# B&R Automation Studio project TrakBasisProject (part 2)

#### Set_Testcases.c
```c
/********************************************************************
 * COPYRIGHT --
 ********************************************************************
 * Program: -
 * Author:
 * Created:
 ********************************************************************
 * Tests for ...
 ********************************************************************/

#include <bur/plctypes.h>

#ifdef _DEFAULT_INCLUDES
#include <AsDefault.h>
#endif

#include "UnitTest.h"

_TEST waitForReadyForPowerOn (void)
{
	TEST_BUSY_CONDITION(0 == gTrakCtrl.Status.ReadyForPowerOn);
	TEST_ASSERT(gTrakCtrl.Status.ReadyForPowerOn);

	TEST_DONE;
}

_TEST waitForCommunicationReady (void)
{
	TEST_BUSY_CONDITION(0 == gTrakCtrl.Status.CommunicationReady);
	TEST_ASSERT(gTrakCtrl.Status.CommunicationReady);

	TEST_DONE;
}

_TEST waitForPLCopenStateDisabled (void)
{
	TEST_ASSERT(gTrakCtrl.Status.PLCopenState.Disabled);

	TEST_DONE;
}

_TEST setPowerOnAndCheckStatus (void)
{
	gTrakCtrl.Command.Power = 1;

	TEST_BUSY_CONDITION(0 == gTrakCtrl.Status.PowerOn);
	TEST_ASSERT(gTrakCtrl.Status.PowerOn);

	TEST_DONE;
}

_TEST waitForPLCopenStateReady (void)
{
	TEST_BUSY_CONDITION(0 == gTrakCtrl.Status.PLCopenState.Ready);
	TEST_ASSERT(gTrakCtrl.Status.PLCopenState.Ready);

	TEST_DONE;
}

_TEST setCommandMoveAbsolute (void)
{
	gTrakCtrl.Command.Move.Absolute = 1;
	gTrakCtrl.Parameter.Position = 0.0;
	gTrakCtrl.Parameter.Speed = 2.0;
	gTrakCtrl.Parameter.Acceleration = 20.0;
	gTrakCtrl.Parameter.Deceleration = 20.0;

	TEST_DONE;
}

_TEST waitForMovementAfterCommandMoveAbsolute (void)
{
	TEST_BUSY_CONDITION(1 == gTrakCtrl.Command.Move.Absolute);
	TEST_BUSY_CONDITION(0 == gTrakCtrl.Status.MovementDetected);
	TEST_ASSERT(gTrakCtrl.Status.MovementDetected);

	TEST_DONE;
}

_TEST waitForMovementAbsoluteStops (void)
{
	TEST_BUSY_CONDITION(1 == gTrakCtrl.Status.MovementDetected);
	TEST_ASSERT(0 == gTrakCtrl.Status.MovementDetected);
	TEST_DONE;
}

_TEST setCommandMoveVelocity (void)
{
	gTrakCtrl.Command.Move.Velocity = 1;
	gTrakCtrl.Parameter.Position = 0.0;
	gTrakCtrl.Parameter.Speed = 2.0;
	gTrakCtrl.Parameter.Acceleration = 20.0;
	gTrakCtrl.Parameter.Deceleration = 20.0;

	TEST_DONE;
}

_TEST waitForMovementAfterCommandMoveVelocity (void)
{
	TEST_BUSY_CONDITION(1 == gTrakCtrl.Command.Move.Velocity);
	TEST_BUSY_CONDITION(0 == gTrakCtrl.Status.MovementDetected);

	TEST_ASSERT(gTrakCtrl.Status.MovementDetected);

	TEST_DONE;
}

_TEST checkActualSpeedAfterCommandMoveVelocity (void)
{
	TEST_BUSY_CONDITION(2.0 > gTrakCtrl.Status.Shuttle[1].ActVelocity);

	TEST_ASSERT(gTrakCtrl.Status.Shuttle[1].Valid);
	TEST_ASSERT_REAL_WITHIN(0.1, 2.0, gTrakCtrl.Status.Shuttle[1].ActVelocity);
	TEST_ASSERT_EQUAL_STRING("Sector_1", gTrakCtrl.Status.Shuttle[1].ActSector);

	TEST_DONE;
}

_TEST setCommandHalt (void)
{
	gTrakCtrl.Command.Move.Halt = 1;

	TEST_DONE;
}

_TEST waitForMovementStopsAfterCommandHalt (void)
{
	TEST_BUSY_CONDITION(1 == gTrakCtrl.Command.Move.Halt);
	TEST_BUSY_CONDITION(1 == gTrakCtrl.Status.MovementDetected);

	TEST_ASSERT(0 == gTrakCtrl.Status.MovementDetected);
	TEST_ASSERT(gTrakCtrl.Status.Shuttle[1].Valid);
	TEST_ASSERT_EQUAL_REAL(0.0, gTrakCtrl.Status.Shuttle[1].ActVelocity);
	TEST_ASSERT_EQUAL_STRING("Sector_1", gTrakCtrl.Status.Shuttle[1].ActSector);

	TEST_DONE;
}

/*
B+R UnitTest: This is generated code.
Do not edit! Do not move!
Description: UnitTest Testprogramm infrastructure (TestSet).
LastUpdated: 2025-09-17 11:53:31Z
By B+R UnitTest Helper Version: 2.0.0.0
*/
UNITTEST_FIXTURES(fixtures)
{
	new_TestFixture("waitForReadyForPowerOn", waitForReadyForPowerOn),
	new_TestFixture("waitForCommunicationReady", waitForCommunicationReady),
	new_TestFixture("waitForPLCopenStateDisabled", waitForPLCopenStateDisabled),
	new_TestFixture("setPowerOnAndCheckStatus", setPowerOnAndCheckStatus),
	new_TestFixture("waitForPLCopenStateReady", waitForPLCopenStateReady),
	new_TestFixture("setCommandMoveAbsolute", setCommandMoveAbsolute),
	new_TestFixture("waitForMovementAfterCommandMoveAbsolute", waitForMovementAfterCommandMoveAbsolute),
	new_TestFixture("waitForMovementAbsoluteStops", waitForMovementAbsoluteStops),
	new_TestFixture("setCommandMoveVelocity", setCommandMoveVelocity),
	new_TestFixture("waitForMovementAfterCommandMoveVelocity", waitForMovementAfterCommandMoveVelocity),
	new_TestFixture("checkActualSpeedAfterCommandMoveVelocity", checkActualSpeedAfterCommandMoveVelocity),
	new_TestFixture("setCommandHalt", setCommandHalt),
	new_TestFixture("waitForMovementStopsAfterCommandHalt", waitForMovementStopsAfterCommandHalt),
};

UNITTEST_CALLER_COMPLETE_EXPLICIT(Set_Testcases, "Set_Testcases", 0, 0, fixtures, 0, 0, 0);
```

### Library Logical/UnitTest/Libraries/UnitTest (ANSIC, version 6.3.0) - Static library for UnitTest programs written in ANSI C /C++

#### UnitTest.h
```c
/*****************************************************************************
 * COPYRIGHT (C) BERNECKER + RAINER
 *****************************************************************************
 * Library:  UnitTest
 * File:     UnitTest.h
 * Author:   B+R
 *****************************************************************************
 * Description: Static library for UnitTest programs written in ANSI C /C++
 *
 * Add the path "\Logical\TS_UnitTest\Libraries\UnitTest\" to the
 * "Additional include directories" in the tab "Build" (PLC Properties)
 ******************************************************************************/

#ifndef	__UNITTEST_H__
#define	__UNITTEST_H__
#ifdef __cplusplus
extern "C"
{
#endif
#include <bur/plctypes.h>

#ifndef NULL
#define	NULL	0
#endif
#include "include/Test.h"

#include "include/TestCase.h"
#include "include/TestListener.h"
#include "include/TestResult.h"
#include "include/TestCaller.h"

#include "include/AssertImpl.h"
#include "include/HelperMacro.h"
#include "include/utRunner.h"

/* function is a test case */
#define _TEST 			static testStatusEnum

/* function is a setup */
#define _SETUP_TEST 	static testStatusEnum 	setupTest

/* function is a teardown */
#define _TEARDOWN_TEST 	static testStatusEnum 	teardownTest

/* function is a setup for whole test set */
#define _SETUP_SET		static testStatusEnum	setupSet

/* function is a teardown for whole test set */
#define _TEARDOWN_SET 	static testStatusEnum	teardownSet

/* function is a cyclic handler for test set */
#define _CYCLIC_SET		static void 			cyclicSetCaller

/* Skipped test case */
#define SKIP_TEST  		_TEST
/* Skip all test cases of set */
#define SKIP_TEST_SET

/* Dummies for smart edit autocompletion.
See AssertImpl.h for real macros used by the compiler  */
#ifdef _SMART_EDIT_DUMMY_

/* String comparison.
Returns true if the strings are equal. */
BOOL TEST_ASSERT_EQUAL_STRING(char *expected,char  *actual);
/* Wstring comparison.
Returns true if the WSTRINGS are equal. */
BOOL TEST_ASSERT_EQUAL_WSTRING(unsigned short *expected,unsigned short *actual);
 /* Compares two memory blocks.
Returns true if [size] bytes are equal. */
BOOL TEST_ASSERT_EQUAL_MEM(void *expected, void *actual,UDINT size);
/* Compares integer values. Usable for all integer types.
Avoid comparison of unsigned with signed types.
Returns true if they are equal.
Note: If different, values are reported as DINT values in the test report */
BOOL TEST_ASSERT_EQUAL_INT(expected, actual);

/* Compares REAL values with delta = (expected * TEST_FLOAT_PRECISION).
Returns true if (difference <= delta) */
BOOL TEST_ASSERT_EQUAL_REAL(REAL expected,REAL actual);
/* Compares REAL values with explicit delta.
Returns true if (difference <= delta) */
BOOL TEST_ASSERT_REAL_WITHIN(REAL delta, REAL expected, REAL actual);
/* Compares LREAL values with delta = (expected * TEST_DOUBLE_PRECISION).
Returns true if (difference <= delta) */
BOOL TEST_ASSERT_EQUAL_LREAL(LREAL expected,LREAL  actual);
/* Compares LREAL values with explicit delta.
Returns true if (difference <= delta) */
BOOL TEST_ASSERT_LREAL_WITHIN(LREAL delta, LREAL expected, LREAL actual);

/* Compares float values with delta = (expected * TEST_FLOAT_PRECISION).
Returns true if (difference <= delta) */
BOOL TEST_ASSERT_EQUAL_FLOAT(float expected, float actual);
/* Compares float values with explicit delta.
Returns true if (difference <= delta) */
BOOL TEST_ASSERT_FLOAT_WITHIN(float delta, float expected, float actual);
/* Compares double values with delta = (expected * TEST_DOUBLE_PRECISION).
Returns true if (difference <= delta) */
BOOL TEST_ASSERT_EQUAL_DOUBLE(double expected, double actual);
/* Compares double values with explicit delta.
Returns true if (difference <= delta) */
BOOL TEST_ASSERT_DOUBLE_WITHIN(double delta, double expected, double actual);

/* Returns true if pointer is null */
BOOL TEST_ASSERT_NULL(void *pointer);
/* Returns true if pointer is not null */
BOOL TEST_ASSERT_NOT_NULL(void *pointer);
/* Returns true, if condition evals to  true */
BOOL TEST_ASSERT_MESSAGE(condition, char *message);
/* Returns true, if condition evals to  true */
BOOL TEST_ASSERT(condition);

/* Returns always false */
BOOL TEST_FAIL(char *message);

/* Add a note to the test report */
void TEST_INFO(char *message);
/* Add a note with location information to the test report */
void TEST_INFO_POS(char *message);

#ifdef __cplusplus
/* Test if expression throws given exception.
Catches all other exceptions as failure.
Note: Available for C++ only */
void TEST_ASSERT_THROW(expression, type);

/* Fails if expression throws any exceptions.
Note: Available for C++ only*/
void TEST_ASSERT_NO_THROW(expression);
#endif

/* Adds a test function with description to the Testfixture.
See UNITTEST_FIXTURES() */
void new_TestFixture(char *name, _TEST function);

/* Adds a test function with description to the Testfixture.
This test will be skipped
See UNITTEST_FIXTURES() */
void skipTestFixture(char *name, _TEST function);

/* Defines the order of test cases.
Should look like this
UNITTEST_FIXTURES(fixtures)
{
	new_TestFixture("test_1",test_1),
	new_TestFixture("test_2",test_2),
	new_TestFixture("test_3",test_3)
}
*/
void UNITTEST_FIXTURES(fixtures)

/* Standard UnitTest caller without any setup / teardown methods*/
void UNITTEST_CALLER_TEST(caller, char *name, fixtures);

/* Standard UnitTest caller with macro setup / teardown for tests*/
void UNITTEST_CALLER_BASIC(caller, char *name, fixtures);

/* UnitTest caller with macro setup / teardown for tests and test set */
void UNITTEST_CALLER_SET(caller, char *name, fixtures);

/* UnitTest caller with macro setup / teardown for tests and test set and cylic*/
void UNITTEST_CALLER_COMPLETE(caller, char *name, fixtures);

/* UnitTest caller with explicit setup / teardown for suite */
void UNITTEST_CALLER_SET_EXPLICIT(caller,name,setupTest,teardownTest,fixtures, setupSuite, teardownSuite);

/* UnitTest caller with explicit setup / teardown for suite and cylic */
void UNITTEST_CALLER_COMPLETE_EXPLICIT(caller,name,setupTest,teardownTest,fixtures, setupSuite, teardownSuite, cyclicCaller);

/* Adds a test set with description to the fixture of test sets.
See UNITTEST_TESTSET_FIXTURES() */
void new_TestSet(testcaller);

/* Defines the order of test sets.
Should look like this
UNITTEST_TESTSET_FIXTURES(fixtures)
{
	new_TestSet(testSet_1),
	new_TestSet(testSet_2),
	new_TestSet(testSet_3)
}*/
void UNITTEST_TESTSET_FIXTURES(fixtures);

/* Defines the test set list handling structure*/
void UNTITTEST_TESTSET_HANDLER();

#endif /*_SMART_EDIT_DUMMY_*/

/*
 Use to declare Test set for use in list of test sets of test programm
 See usage in autogeneratedFile.c / FixtureOfTestSets.c
*/
#define UNITTEST_TESTSET_DECLARATION 	extern const TestCaller

/* Default factor for precision used to test if REAL / float values  are equal.
(0.00001f) */
#define TEST_FLOAT_PRECISION 	(0.00001f)
/* Default factor for precision used to test if LREAL / double values  are equal.
(1e - 12f) */
#define TEST_DOUBLE_PRECISION 	(1e-12f)

#if (__GNUC__ != 11) || (__GNUC_MINOR__ != 3) || (__GNUC_PATCHLEVEL__ != 0)
#error UnitTest is compiled with GCC version 11.3.0. To use UnitTest switch GCC version to 11.3.0 or import a different solution package
#endif

#define UNIT_TEST_LIBRARY_VERSION  			"6.3.0"

#ifdef __cplusplus
};
#endif

#include "include/asserts.hpp"

#endif/*__UNITTEST_H__*/
```

#### AssertImpl.c
```c
/*
 * COPYRIGHT AND PERMISSION NOTICE
 *
 * Copyright (c) 2003 Embedded Unit Project
 *
 * All rights reserved.
 *
 * Permission is hereby granted, free of charge, to any person obtaining
 * a copy of this software and associated documentation files (the
 * "Software"), to deal in the Software without restriction, including
 * without limitation the rights to use, copy, modify, merge, publish,
 * distribute, and/or sell copies of the Software, and to permit persons
 * to whom the Software is furnished to do so, provided that the above
 * copyright notice(s) and this permission notice appear in all copies
 * of the Software and that both the above copyright notice(s) and this
 * permission notice appear in supporting documentation.
 *
 * THE SOFTWARE IS PROVIDED "AS IS", WITHOUT WARRANTY OF ANY KIND,
 * EXPRESS OR IMPLIED, INCLUDING BUT NOT LIMITED TO THE WARRANTIES OF
 * MERCHANTABILITY, FITNESS FOR A PARTICULAR PURPOSE AND NONINFRINGEMENT
 * OF THIRD PARTY RIGHTS. IN NO EVENT SHALL THE COPYRIGHT HOLDER OR
 * HOLDERS INCLUDED IN THIS NOTICE BE LIABLE FOR ANY CLAIM, OR ANY
 * SPECIAL INDIRECT OR CONSEQUENTIAL DAMAGES, OR ANY DAMAGES WHATSOEVER
 * RESULTING FROM LOSS OF USE, DATA OR PROFITS, WHETHER IN AN ACTION OF
 * CONTRACT, NEGLIGENCE OR OTHER TORTIOUS ACTION, ARISING OUT OF OR IN
 * CONNECTION WITH THE USE OR PERFORMANCE OF THIS SOFTWARE.
 *
 * Except as contained in this notice, the name of a copyright holder
 * shall not be used in advertising or otherwise to promote the sale,
 * use or other dealings in this Software without prior written
 * authorization of the copyright holder.
 *
 * $Id: AssertImpl.c,v 1.5 2004/02/10 16:15:25 arms22 Exp $
 */

#include "include/AssertImpl.h"

#include "src/embunit/stdImpl_c.h"

#define FALSE 0
#define TRUE  1

/*
 * Note: Less than 255,  a char is used as counter
*/
#define ASSERT_STRING_BUFFER_MAX	200
#define ASSERT_NUMBER_BUFFER_MAX	100

BOOL assertCondition(BOOL condition, const char *message, unsigned  long line, const char *file)
{
	if (condition)
	{
		addPassed("", line, file);
		return TRUE;
	}
	else
	{
		addFailure(message, line, file);
		return FALSE;
	}
}

BOOL assertImplementationInt(int expected, int actual, unsigned  long line, const char *file)
{

	if (expected == actual)
	{
		addPassed("", line, file);
		return TRUE;
	}
	else
	{
		char buffer[ASSERT_NUMBER_BUFFER_MAX];	/*"exp -2147483647 was -2147483647"*/
		char numbuf[12];	/*32bit int decimal maximum column is 11 (-2147483647~2147483647)*/

		stdimpl_strcpy(buffer, "exp ");

		{
			stdimpl_itoa(expected, numbuf, 10);
			stdimpl_strncat(buffer, numbuf, 11);
		}

		stdimpl_strcat(buffer, " was ");

		{
			stdimpl_itoa(actual, numbuf, 10);
			stdimpl_strncat(buffer, numbuf, 11);
		}

		addFailure(buffer, line, file);
		return FALSE;
	}
}

BOOL assertImplementationMem(void *expected, void  *actual, unsigned long  size, unsigned  long line, const char *file)
{
	signed short compare = 0;
	char buffer[ASSERT_STRING_BUFFER_MAX];
	if(expected && actual && size)
	{

		compare = stdimpl_memcmp(expected,actual,size);
		if (0 == compare)
		{
			addPassed("", line, file);
			return TRUE;
		}
		else
		{

			char numbuf[12];	/*32bit int decimal maximum column is 11 (-2147483647~2147483647)*/

			stdimpl_strcpy(buffer, "Result of memory comparison was ");

			{
				stdimpl_itoa(compare, numbuf, 10);
				stdimpl_strncat(buffer, numbuf, 11);
			}

			addFailure(buffer, line, file);
			return FALSE;
		}

	}
	else
	{
		if(!size)
		{
			stdimpl_strcpy(buffer, "Invalid size for comparison ");
			addFailure(buffer, line, file);
			return FALSE;
		}
		else if (!actual)
		{
			stdimpl_strcpy(buffer, "acutal value was a nullpointer ");
			addFailure(buffer, line, file);
			return FALSE;
		}
		else /*(!expected)*/
		{
			stdimpl_strcpy(buffer, "expected value was a nullpointer ");
			addFailure(buffer, line, file);
			return FALSE;
		}
	}
}

BOOL assertImplementationCStr(const char *expected, const char *actual, unsigned  long line, const char *file)
{
	if (expected && actual && (stdimpl_strcmp(expected,actual)==0) )
	{
		addPassed("", line, file);
		return TRUE;
	}
	else
	{
		char buffer[ASSERT_STRING_BUFFER_MAX];
#define exp_act_limit ((ASSERT_STRING_BUFFER_MAX- 15 - 1)/2)/*	"exp'' was''" = 11 byte	*/
		int el;
		int al;

		if (expected)
		{
			el = stdimpl_strlen(expected);
		}
		else
		{
			el = 4;
			expected = "null";
		}

		if (actual)
		{
			al = stdimpl_strlen(actual);
		}
		else
		{
			al = 4;
			actual = "null";
		}
		if (el > exp_act_limit)
		{
			if (al > exp_act_limit)
			{
				al = exp_act_limit;
				el = exp_act_limit;
			}
			else
			{
				int w = exp_act_limit + (exp_act_limit - al);
				if (el > w)
				{
					el = w;
				}
			}
		}
		else
		{
			int w = exp_act_limit + (exp_act_limit - el);
			if (al > w)
			{
				al = w;
			}
		}
		stdimpl_strcpy(buffer, "exp \"");
		stdimpl_strncat(buffer, expected, el);
		stdimpl_strcat(buffer, "\" was \"");
		stdimpl_strncat(buffer, actual, al);
		stdimpl_strcat(buffer, "\"");

		addFailure(buffer, line, file);
		return FALSE;
	}
#undef exp_act_limit
}

/*
 * Author: 		B&R
 * Added: 		September 04, 2012
 *
 */
BOOL assertImplementationDoublesWithin(const double delta,
	const double expected,
	const double actual,
	unsigned long line, const char *file)
{
	char buffer[ASSERT_NUMBER_BUFFER_MAX];	/*"exp -2147483647 was -2147483647"*/
	char numbuf[22];	/*32bit int decimal maximum column is 11 (-2147483647~2147483647)*/

	double diff = actual - expected;
	double pos_delta = delta;

	if (diff < 0)
	{
		diff = 0.0f - diff;
	}
	if (pos_delta < 0)
	{
		pos_delta = 0.0f - pos_delta;
	}

	if (pos_delta < diff)
	{
		stdimpl_strcpy(buffer, "exp ");
		stdimpl_dtoa(expected, &numbuf[0], sizeof(numbuf));
		stdimpl_strncat(buffer, numbuf, 11);

		stdimpl_strcat(buffer, " was ");
		stdimpl_dtoa(actual, &numbuf[0], sizeof(numbuf));
		stdimpl_strncat(buffer, numbuf, 11);

		addFailure(buffer, line, file);
		return FALSE;
	}
	else
	{
		addPassed("", line, file);
		return TRUE;
	}
}

/*
 * Author: 		B&R
 * Added: 		September 04, 2012
 *
 */
BOOL assertImplementationFloatsWithin(const float delta,
	const float expected,
	const float actual,
	unsigned long line, const char *file)
{
	char buffer[ASSERT_NUMBER_BUFFER_MAX];	/*"exp -2147483647 was -2147483647"*/
	char numbuf[22];	/*32bit int decimal maximum column is 11 (-2147483647~2147483647)*/

	float diff = actual - expected;
	float pos_delta = delta;

	if (diff < 0)
	{
		diff = 0.0f - diff;
	}
	if (pos_delta < 0)
	{
		pos_delta = 0.0f - pos_delta;
	}

	if (pos_delta < diff)
	{
		stdimpl_strcpy(buffer, "exp ");
		stdimpl_ftoa(expected, &numbuf[0], sizeof(numbuf));
		stdimpl_strncat(buffer, numbuf, 11);

		stdimpl_strcat(buffer, " was ");
		stdimpl_ftoa(actual, &numbuf[0], sizeof(numbuf));
		stdimpl_strncat(buffer, numbuf, 11);

		addFailure(buffer, line, file);
		return FALSE;
	}
	else
	{
		addPassed("", line, file);
		return TRUE;
	}
}

/*
 * Author: 		B&R
 * Added: 		August 21, 2012
 * Modified: 	October 09, 2012
 *
 * Prints dezimal value of the WSTRING characters
 */
BOOL assertImplementationWStr(const unsigned short *expected, const unsigned short *actual, unsigned long line, const char *file)
{
	if (expected && actual && (stdimpl_Wstrcmp(expected,actual)==0))
	{
		addPassed("", line, file);
		return TRUE;
	}
	else
	{

		char buffer[ASSERT_STRING_BUFFER_MAX*2];

#define exp_act_limit ((ASSERT_STRING_BUFFER_MAX- 15 - 1)/2 / sizeof(unsigned short))/*	"exp'' was''" = 11 byte	*/
#define MAX_LEN 6 /* "65535 " */
		int el;
		int al;

		if (expected)
		{
			el = MAX_LEN * (sizeof(unsigned short) * stdimpl_Wstrlen(expected));
		}
		else
		{
			el = 4;
			/* will be append later */
		}

		if (actual)
		{
			al = MAX_LEN * (sizeof(unsigned short) * stdimpl_Wstrlen(actual));
		}
		else
		{
			al = 4;
			/* will be append later */
		}
		if (el > exp_act_limit)
		{
			if (al > exp_act_limit)
			{
				al = exp_act_limit;
				el = exp_act_limit;
			}
			else
			{
				int w = exp_act_limit + (exp_act_limit - al);
				if (el > w)
				{
					el = w;
				}
			}
		}
		else
		{
			int w = exp_act_limit + (exp_act_limit - el);
			if (al > w)
			{
				al = w;
			}
		}
		stdimpl_strcpy(buffer, "exp \"");
		if(expected)
			stdimpl_Wstrncat(buffer, expected, el/(sizeof(unsigned short)) );
		else
			stdimpl_strcat(buffer, "null");
		stdimpl_strcat(buffer, "\" was \"");
		if(actual)
			stdimpl_Wstrncat(buffer, actual, al/(sizeof(unsigned short)) );
		else
			stdimpl_strcat(buffer, "null");
		stdimpl_strcat(buffer, "\"");

		addFailure(buffer, line, file);
		return FALSE;
	}
#undef exp_act_limit
}
```

#### stdImpl_c.h
```c
/*
 * COPYRIGHT AND PERMISSION NOTICE
 *
 * Copyright (c) 2003 Embedded Unit Project
 *
 * All rights reserved.
 *
 * Permission is hereby granted, free of charge, to any person obtaining
 * a copy of this software and associated documentation files (the
 * "Software"), to deal in the Software without restriction, including
 * without limitation the rights to use, copy, modify, merge, publish,
 * distribute, and/or sell copies of the Software, and to permit persons
 * to whom the Software is furnished to do so, provided that the above
 * copyright notice(s) and this permission notice appear in all copies
 * of the Software and that both the above copyright notice(s) and this
 * permission notice appear in supporting documentation.
 *
 * THE SOFTWARE IS PROVIDED "AS IS", WITHOUT WARRANTY OF ANY KIND,
 * EXPRESS OR IMPLIED, INCLUDING BUT NOT LIMITED TO THE WARRANTIES OF
 * MERCHANTABILITY, FITNESS FOR A PARTICULAR PURPOSE AND NONINFRINGEMENT
 * OF THIRD PARTY RIGHTS. IN NO EVENT SHALL THE COPYRIGHT HOLDER OR
 * HOLDERS INCLUDED IN THIS NOTICE BE LIABLE FOR ANY CLAIM, OR ANY
 * SPECIAL INDIRECT OR CONSEQUENTIAL DAMAGES, OR ANY DAMAGES WHATSOEVER
 * RESULTING FROM LOSS OF USE, DATA OR PROFITS, WHETHER IN AN ACTION OF
 * CONTRACT, NEGLIGENCE OR OTHER TORTIOUS ACTION, ARISING OUT OF OR IN
 * CONNECTION WITH THE USE OR PERFORMANCE OF THIS SOFTWARE.
 *
 * Except as contained in this notice, the name of a copyright holder
 * shall not be used in advertising or otherwise to promote the sale,
 * use or other dealings in this Software without prior written
 * authorization of the copyright holder.
 *
 * $Id: stdImpl.c,v 1.3 2004/02/10 16:15:25 arms22 Exp $
 */

#include "UtMgr.h"

static char *stdimpl_strcpy(char *dst, const char *src)
{
	char *start = dst;
	char c;
	do
	{
		c = *src;
		*dst = c;
		src++;
		dst++;
	}
	while (c);
	return start;
}
/* currently not used */
#if 0
/*
 * Author: 		B&R
 * Added: 		December 20, 2012
 */
static char *stdimpl_strrchr(char *src, const char chr)
{
	char *pos = 0;
	char c;
	do
	{
		c = *src;
		if(chr == c)
		{
			pos = src;
		}
		src++;
	}
	while (c);
	return pos;
}
/*
 * Author: 		B&R
 * Added: 		December 20, 2012
 */
static char *stdimpl_memcpy(char *dst, const char *src, unsigned long len)
{
	char *start = dst;
	char c;
	unsigned long i = 0;
	for(i= 0; i<len; i++)
	{
		c = *src;
		*dst = c;
		src++;
		dst++;
	}
	return start;
}
#endif

static char *stdimpl_strcat(char *dst, const char *src)
{
	char *start = dst;
	char c;
	do
	{
		c = *dst;
		dst++;
	}
	while (c);
	dst--;
	do
	{
		c = *src;
		*dst = c;
		src++;
		dst++;
	}
	while (c);
	return start;
}

static char *stdimpl_strncat(char *dst, const char *src,unsigned int count)
{
	char *start = dst;
	char c;
	do
	{
		c = *dst;
		dst++;
	}
	while (c);
	dst--;
	if (count)
	{
		do
		{
			c = *src;
			*dst = c;
			src++;
			dst++;
			count--;
		}
		while (c && count);
		*dst = '\0';
	}
	return start;
}

static int stdimpl_strlen(const char *str)
{
	const char *estr = str;
	char c;
	do
	{
		c = *estr;
		estr++;
	}
	while (c);
	return ((int)(estr - str - 1));
}

static int stdimpl_strcmp(const char *s1, const char *s2)
{
	char c1,c2;
	do
	{
		c1 = *s1++;
		c2 = *s2++;
	}
	while ((c1) && (c2) && (c1==c2));
	return c1 - c2;
}

static char *_xtoa(unsigned long v,char *string, int r, int is_neg)
{
	char *start = string;
	char buf[33],*p;

	p = buf;

	do
	{
		*p++ = "0123456789abcdef"[(v % r) & 0xf];
	}
	while (v /= r);

	if (is_neg)
	{
		*p++ = '-';
	}

	do
	{
		*string++ = *--p;
	}
	while (buf != p);

	*string = '\0';

	return start;
}

static char *stdimpl_itoa(int v,char *string,int r)
{
	if ((r == 10) && (v < 0))
	{
		return _xtoa((unsigned long)(-v), string, r, 1);
	}
	return _xtoa((unsigned long)(v), string, r, 0);
}

/*
 * Author: 		B&R
 * Added: 		August 21, 2012
 * Modified: 	October 09, 2012
 */
static char *stdimpl_Wstrncat(char *dst, const unsigned short *src,unsigned int count)
{
	char *start = dst;

	unsigned short c;

	do
	{
		c = *dst;
		dst++;
	}
	while (c);
	dst--;
	if (count)
	{
		do
		{
			c = *src;

			dst += 	stdimpl_strlen(stdimpl_itoa(c, dst, 10));
			*dst = ' ';
			dst++;
			src++;
			count--;
		}
		while (c && count);
		*dst = '\0';
	}
	return start;
}

/*
 * Author: 		B&R
 * Added: 		August 21, 2012
 * Modified: 	October 09, 2012
 */
static int stdimpl_Wstrlen(const unsigned short *str)
{
	const unsigned short *estr = str;
	unsigned short c;
	do
	{
		c = *estr;
		estr++;
	}
	while (c);
	return ((int)(estr - str - 1));
}

/*
 * Author: 		B&R
 * Added: 		August 21, 2012
 * Modified: 	October 09, 2012
 */
static int stdimpl_Wstrcmp(const unsigned short *s1, const unsigned short *s2)
{
	unsigned short c1,c2;
	do
	{
		c1 = *s1++;
		c2 = *s2++;
	}
	while ((c1) && (c2) && (c1==c2));
	return c1 - c2;
}

static char *stdimpl_ftoa(float v,char *string, unsigned long len)
{
	/*iec_double2str(v, sizeof(float), string, len);*/
	return	(char *)UtMgrHelperFtoa(v, sizeof(float),(unsigned long) string, len);

}

static char *stdimpl_dtoa(double v,char *string, unsigned long len)
{
	/*iec_double2str(v, sizeof(double), string, len);*/
	return	(char *)UtMgrHelperFtoa(v, sizeof(double), (unsigned long) string, len);

}

static char stdimpl_memcmp(const void *s1, const void *s2, unsigned long len)
{
	char c1,c2;
	unsigned long i = 0;
	for(i = 0; i < len; i++)
	{
		c1 = *(char *)s1++;
		c2 = *(char *)s2++;
		if(c1 != c2)
			return c1 - c2;
	}
	return c1 - c2;
}
```

#### TestResult.c
```c
/*
 * COPYRIGHT AND PERMISSION NOTICE
 *
 * Copyright (c) 2003 Embedded Unit Project
 *
 * All rights reserved.
 *
 * Permission is hereby granted, free of charge, to any person obtaining
 * a copy of this software and associated documentation files (the
 * "Software"), to deal in the Software without restriction, including
 * without limitation the rights to use, copy, modify, merge, publish,
 * distribute, and/or sell copies of the Software, and to permit persons
 * to whom the Software is furnished to do so, provided that the above
 * copyright notice(s) and this permission notice appear in all copies
 * of the Software and that both the above copyright notice(s) and this
 * permission notice appear in supporting documentation.
 *
 * THE SOFTWARE IS PROVIDED "AS IS", WITHOUT WARRANTY OF ANY KIND,
 * EXPRESS OR IMPLIED, INCLUDING BUT NOT LIMITED TO THE WARRANTIES OF
 * MERCHANTABILITY, FITNESS FOR A PARTICULAR PURPOSE AND NONINFRINGEMENT
 * OF THIRD PARTY RIGHTS. IN NO EVENT SHALL THE COPYRIGHT HOLDER OR
 * HOLDERS INCLUDED IN THIS NOTICE BE LIABLE FOR ANY CLAIM, OR ANY
 * SPECIAL INDIRECT OR CONSEQUENTIAL DAMAGES, OR ANY DAMAGES WHATSOEVER
 * RESULTING FROM LOSS OF USE, DATA OR PROFITS, WHETHER IN AN ACTION OF
 * CONTRACT, NEGLIGENCE OR OTHER TORTIOUS ACTION, ARISING OUT OF OR IN
 * CONNECTION WITH THE USE OR PERFORMANCE OF THIS SOFTWARE.
 *
 * Except as contained in this notice, the name of a copyright holder
 * shall not be used in advertising or otherwise to promote the sale,
 * use or other dealings in this Software without prior written
 * authorization of the copyright holder.
 *
 * $Id: TestResult.c,v 1.4 2004/02/10 16:19:29 arms22 Exp $
 */
#include "src/utOther.h"
#include "include/Test.h"
#include "include/TestListener.h"
#include "include/TestResult.h"

/*
 * Author: 		B&R
 * Modified: 	October   09, 2012
*/
void TestResult_init(TestResult *self,TestListner *listner)
{
	if(!self)
		return;

	self->runCount = 0;
	self->failureCount = 0;
	self->passedCount = 0;
	self->summarizedCount = 0;
	self->abortCount = 0;
	self->suceessedTestCount = 0;
	self->skippedTestCount = 0;
	self->infoCount = 0;
	self->listener = listner;

}

void TestResult_startTest(TestResult *self,Test *test)
{
	if(!self)
		return;
	self->runCount++;

	if (self->listener)
	{
		TestListener_doLog(self->listener, test, 0, 0, 0, utProf_Ev_Name_Test_Start);
		TestListner_startTest(self->listener, test);
	}
}

void TestResult_endTest(TestResult *self,Test *test)
{
	if(!self)
		return;

	if (self->listener)
	{
		TestListener_doLog(self->listener, test, 0, 0, 0, utProf_Ev_Name_Test_End);
		TestListner_endTest(self->listener, test);
	}
}

void TestResult_skipTest(TestResult *self,Test *test)
{
	if(!self)
		return;
	self->runCount++;
	if (self->listener)
	{
		TestListener_doLog(self->listener, test, 0, 0, 0, utProf_Ev_Skipped);
		TestListner_skippedTest(self->listener, test);
	}
}

/*
 * Author: 		B&R
 * Modified: 	October   09, 2012
*/
void TestResult_addFailure(TestResult *self,Test *test,const char *msg,unsigned long line,const char *file)
{
	if(!self)
		return;
	self->summarizedCount++;
	self->failureCount++;
	if (self->listener)
	{
		TestListener_doLog(self->listener, test, msg, line, file, utProf_Ev_MsgFail);
		TestListner_addFailure(self->listener, test, msg, line, file);
	}
}

/*
 * Author: 		B&R
 * Added: 		October   09, 2012
*/
void TestResult_addPassed(TestResult *self,Test *test,const char *msg,unsigned long line,const char *file)
{
	if(!self )
		return;

	self->summarizedCount++;
	self->passedCount++;
	/*! \note changed: add passed wird nun auch aufgerufen --> interessant für Json*/
	if (self->listener)
	{
		TestListener_doLog(self->listener, test, msg, line, file, utProf_Ev_MsgPass);
		TestListner_addPassed(self->listener, test, msg, line, file);
	}
}

/*
 * Author: 		B&R
 * Added: 		October   23, 2012
*/
void TestResult_addInfo(TestResult *self,Test *test,const char *msg,unsigned long line,const char *file)
{
	if(!self )
		return;
	self->infoCount++;

	if (self->listener)
	{
		TestListener_doLog(self->listener, test, msg, line, file, utProf_Ev_MsgInfo);
		TestListner_addInfo(self->listener, test, msg, line, file);
	}
}

void TestResult_addAbort(TestResult *self,Test *test,const char *msg,unsigned long line,const char *file)
{
	if(!self )
		return;
	self->abortCount++;
	if (self->listener)
	{
		TestListener_doLog(self->listener, test, msg, line, file, utProf_Ev_MsgAbort);
		TestListner_addAbort(self->listener, test, msg, line, file);
	}
}
```

#### TestCaller.c
```c
/*
 * COPYRIGHT AND PERMISSION NOTICE
 *
 * Copyright (c) 2003 Embedded Unit Project
 *
 * All rights reserved.
 *
 * Permission is hereby granted, free of charge, to any person obtaining
 * a copy of this software and associated documentation files (the
 * "Software"), to deal in the Software without restriction, including
 * without limitation the rights to use, copy, modify, merge, publish,
 * distribute, and/or sell copies of the Software, and to permit persons
 * to whom the Software is furnished to do so, provided that the above
 * copyright notice(s) and this permission notice appear in all copies
 * of the Software and that both the above copyright notice(s) and this
 * permission notice appear in supporting documentation.
 *
 * THE SOFTWARE IS PROVIDED "AS IS", WITHOUT WARRANTY OF ANY KIND,
 * EXPRESS OR IMPLIED, INCLUDING BUT NOT LIMITED TO THE WARRANTIES OF
 * MERCHANTABILITY, FITNESS FOR A PARTICULAR PURPOSE AND NONINFRINGEMENT
 * OF THIRD PARTY RIGHTS. IN NO EVENT SHALL THE COPYRIGHT HOLDER OR
 * HOLDERS INCLUDED IN THIS NOTICE BE LIABLE FOR ANY CLAIM, OR ANY
 * SPECIAL INDIRECT OR CONSEQUENTIAL DAMAGES, OR ANY DAMAGES WHATSOEVER
 * RESULTING FROM LOSS OF USE, DATA OR PROFITS, WHETHER IN AN ACTION OF
 * CONTRACT, NEGLIGENCE OR OTHER TORTIOUS ACTION, ARISING OUT OF OR IN
 * CONNECTION WITH THE USE OR PERFORMANCE OF THIS SOFTWARE.
 *
 * Except as contained in this notice, the name of a copyright holder
 * shall not be used in advertising or otherwise to promote the sale,
 * use or other dealings in this Software without prior written
 * authorization of the copyright holder.
 *
 * $Id: TestCaller.c,v 1.6 2004/02/10 16:19:29 arms22 Exp $
 */
#include "src/utOther.h"
#include "include/Test.h"
#include "include/TestResult.h"

#include "include/TestListener.h"
#include "include/TestCase.h"
#include "include/TestCaller.h"

#include "src/embunit/profiling.h"

extern TestResult *result_;
extern TestCase *self_;

const char *TestCaller_name(TestCaller *self)
{
	return self->name;
}

TestCase cs = new_TestCase(0,0,0,0);

int loopCounter = 0;

char TestCaller_run(TestCaller *self,TestResult *result)
{
	switch(self->state)
	{
		case stateStart:
			{
				self->abort = 0;
				TestListener_doLog(result->listener, self, 0,0,0,utProf_Ev_Name_Set_Start);
				loopCounter  = 0;
				self->state = stateSetup;

				if(0 == (self->mode) )/* Skip */
				{

					while(loopCounter < self->numberOfFixtuers)
					{
						cs.isa = (TestImplement *)&TestCaseImplement;
						cs.abort = 0;

						cs.setUp	= self->setUp;
						cs.tearDown	= self->tearDown;

						cs.name		= self->fixtuers[loopCounter].name;
						cs.runTest	= self->fixtuers[loopCounter].test;

						cs.mode = self->fixtuers[loopCounter].mode;

						TestResult 	*wr = result_;	/*push*/
						TestCase 	*ws = self_;	/*push*/

						result_ 	= result;
						self_ 		= (TestCase *)self; /* Attention TestCase != TestCaller in some structure members! */

						TestResult_skipTest(result,(Test*)&cs);

						result_ 	= wr;	/*pop*/
						self_ 		= ws;	/*pop*/

						loopCounter++;
					}

					self->state = stateDefault;
					break;
				}

			}
		case stateSetup:
			{
				if(self->setUpSuite)
				{
					TestResult 	*wr = result_;	/*push*/
					TestCase 	*ws = self_;	/*push*/

					result_ 	= result;
					self_ 		= (TestCase *)self; /* Attention TestCase != TestCaller in some structure members! */
					TestListener_doLog(result->listener, self, 0,0,0,utProf_Ev_SetSetup_Start);
					switch(self->setUpSuite())
					{
						case ut_BUSY:
							break;
						case ut_DONE:
							self->state = stateRun;
							break;
						case ut_ABORT:
							TestListener_doLog(result->listener, self, 0,0,0,utProf_Ev_Abort);
							self->state = stateTearDown;
							self->abort = 1;
							break;
					}
					TestListener_doLog(result->listener, self, 0,0,0,utProf_Ev_SetSetup_End);
					if(self->cyclicSetCaller)
					{
						TestListener_doLog(result->listener, self, 0,0,0,utProf_Ev_SetCylic_Start);
						self->cyclicSetCaller();
						TestListener_doLog(result->listener, self, 0,0,0,utProf_Ev_SetCylic_End);
					}
					result_ 	= wr;	/*pop*/
					self_ 		= ws;	/*pop*/

					break;

				}
				else
				{
					self->state = stateRun;
				}

			}
		case stateRun:
			{
				if(!self->numberOfFixtuers)
				{
					self->state= stateTearDown;

				}
				else
				{
					if(stateStart == cs.state  )
					{
						/* init test */
						cs.isa = (TestImplement *)&TestCaseImplement;
						cs.abort = 0;

						cs.setUp	= self->setUp;
						cs.tearDown	= self->tearDown;

						cs.name		= self->fixtuers[loopCounter].name;
						cs.runTest	= self->fixtuers[loopCounter].test;

						cs.mode = self->fixtuers[loopCounter].mode;

						if( 0 == cs.mode) /* skip this test */
						{
							TestResult 	*wr = result_;	/*push*/
							TestCase 	*ws = self_;	/*push*/

							result_ 	= result;
							self_ 		= (TestCase *)self; /* Attention TestCase != TestCaller in some structure members! */

							TestResult_skipTest(result,(Test*)&cs);

							result_ 	= wr;	/*pop*/
							self_ 		= ws;	/*pop*/

							cs.state =	stateDefault;
						}

					}
					if( 1 == cs.mode) /*  this test is not skipped */
					{
						TestListener_doLog(result->listener, self, 0,0,0,utProf_Ev_Fixture_Start);
						/*run test*/
						Test_run(&cs,result);
						TestListener_doLog(result->listener, self, 0,0,0,utProf_Ev_Fixture_End);

						if(self->cyclicSetCaller)
						{

							TestResult 	*wr = result_;	/*push*/
							TestCase *ws = self_;	/*push*/

							result_ 	= result;
							self_ 		= (TestCase *)self; /* Attention TestCase != TestCaller in some structure members! */

							TestListener_doLog(result->listener, self, 0,0,0,utProf_Ev_SetCylic_Start);

							self->cyclicSetCaller();

							TestListener_doLog(result->listener, self, 0,0,0,utProf_Ev_SetCylic_End);

							result_ 	= wr;	/*pop*/
							self_ 		= ws;	/*pop*/

						}
					}
					/** to go to next test */
					if(stateDefault == cs.state)
					{
						cs.state = stateStart;

						if(cs.abort)
						{
							self->state = stateTearDown;
							self->abort = 1;

							TestListener_doLog(result->listener, self, 0,0,0,utProf_Ev_Abort);
						}
						else
						{
							loopCounter++;
							/* Last test */
							if(loopCounter == self->numberOfFixtuers )
							{
								loopCounter  = 0;
								self->state = stateTearDown;
							}

						}
					}

				}
				break;

			}
		case stateTearDown:
			{
				if(self->tearDownSuite)
				{
					TestResult 	*wr = result_;	/*push*/
					TestCase *ws = self_;	/*push*/

					result_ 	= result;
					self_ 		= (TestCase *)self; /* Attention TestCase != TestCaller in some structure members! */
					switch(self->tearDownSuite())
					{
						case ut_BUSY:
							break;
						case ut_DONE:
							self->state = stateEnd;
							break;
						case ut_ABORT:
							self->state = stateEnd;
							self->abort = 1;
							TestListener_doLog(result->listener, self, 0,0,0,utProf_Ev_Abort);

							break;
					}
					if(self->cyclicSetCaller)
					{
						TestListener_doLog(result->listener, self, 0,0,0,utProf_Ev_SetCylic_Start);
						self->cyclicSetCaller();
						TestListener_doLog(result->listener, self, 0,0,0,utProf_Ev_SetCylic_End);
					}
					result_ 	= wr;	/*pop*/
					self_ 		= ws;	/*pop*/

					if(stateEnd != self->state)
					{
						break;
					}
				}
				else
				{
					self->state = stateEnd;
				}

			}
		case stateEnd:
		case stateDefault:
		default:
			{
				TestListener_doLog(result->listener, self, 0,0,0,utProf_Ev_Name_Set_End);
				self->state = stateDefault;
				return ut_DONE;
			}
	}

	return ut_BUSY;
}

int TestCaller_countTestCases(TestCaller *self)
{
	return self->numberOfFixtuers;
}

const TestImplement TestCallerImplement =
	{
	(TestNameFunction)			TestCaller_name,
	(TestRunFunction)			TestCaller_run,
	(TestCountTestCasesFunction)TestCaller_countTestCases,
	};
```

#### TestCase.c
```c
/*
 * COPYRIGHT AND PERMISSION NOTICE
 *
 * Copyright (c) 2003 Embedded Unit Project
 *
 * All rights reserved.
 *
 * Permission is hereby granted, free of charge, to any person obtaining
 * a copy of this software and associated documentation files (the
 * "Software"), to deal in the Software without restriction, including
 * without limitation the rights to use, copy, modify, merge, publish,
 * distribute, and/or sell copies of the Software, and to permit persons
 * to whom the Software is furnished to do so, provided that the above
 * copyright notice(s) and this permission notice appear in all copies
 * of the Software and that both the above copyright notice(s) and this
 * permission notice appear in supporting documentation.
 *
 * THE SOFTWARE IS PROVIDED "AS IS", WITHOUT WARRANTY OF ANY KIND,
 * EXPRESS OR IMPLIED, INCLUDING BUT NOT LIMITED TO THE WARRANTIES OF
 * MERCHANTABILITY, FITNESS FOR A PARTICULAR PURPOSE AND NONINFRINGEMENT
 * OF THIRD PARTY RIGHTS. IN NO EVENT SHALL THE COPYRIGHT HOLDER OR
 * HOLDERS INCLUDED IN THIS NOTICE BE LIABLE FOR ANY CLAIM, OR ANY
 * SPECIAL INDIRECT OR CONSEQUENTIAL DAMAGES, OR ANY DAMAGES WHATSOEVER
 * RESULTING FROM LOSS OF USE, DATA OR PROFITS, WHETHER IN AN ACTION OF
 * CONTRACT, NEGLIGENCE OR OTHER TORTIOUS ACTION, ARISING OUT OF OR IN
 * CONNECTION WITH THE USE OR PERFORMANCE OF THIS SOFTWARE.
 *
 * Except as contained in this notice, the name of a copyright holder
 * shall not be used in advertising or otherwise to promote the sale,
 * use or other dealings in this Software without prior written
 * authorization of the copyright holder.
 *
 * $Id: TestCase.c,v 1.6 2004/02/10 16:19:29 arms22 Exp $
 */
#include "src/utOther.h"
#include "include/Test.h"
#include "include/TestCase.h"
#include "include/TestResult.h"

#include "include/TestListener.h"
#include "src/embunit/profiling.h"

TestResult *result_;
TestCase *self_;

const char *TestCase_name(TestCase *self)
{
	return self->name;
}

void TestCase_run(TestCase *self,TestResult *result)
{
	switch(self->state)
	{
		case stateStart:
		{
			TestResult_startTest(result, (Test *)self);
			self->state = stateSetup;
		}
		case stateSetup:
		{
			if (self->setUp)
			{
				TestResult 	*wr = result_;	/*push*/
				TestCase *ws = self_;	/*push*/

				result_ 	= result;
				self_ 		= self;
				TestListener_doLog(result->listener, self, 0,0,0,utProf_Ev_TestSetup_Start);
				switch(self->setUp())
				{
					case ut_BUSY:
						break;
					case ut_DONE:
						self->state = stateRun;
						break;
					case ut_ABORT:
						TestListener_doLog(result->listener, self, 0,0,0,utProf_Ev_Abort);
						self->state = stateTearDown;
						self->abort = 1;
						break;
				}
				TestListener_doLog(result->listener, self, 0,0,0,utProf_Ev_TestSetup_End);
				result_ 	= wr;	/*pop*/
				self_ 		= ws;	/*pop*/
				break;
			}
			else
			{
				self->state = stateRun;
			}

		}

		case stateRun:
		{
			if( self->runTest )
			{
				TestResult 	*wr = result_;	/*push*/
				TestCase *ws = self_;	/*push*/

				result_ 	= result;
				self_ 		= self;

				TestListener_doLog(result->listener, self, 0,0,0,utProf_Ev_TestCase_Start);
				switch(self->runTest())
				{
					case ut_BUSY:
						break;
					case ut_DONE:
						self->state = stateTearDown;
						break;
					case ut_ABORT:
						TestListener_doLog(result->listener, self, 0,0,0,utProf_Ev_Abort);
						self->state = stateTearDown;
						self->abort = 1;
						break;
				}
				TestListener_doLog(result->listener, self, 0,0,0,utProf_Ev_TestCase_End);
				result_ 	= wr;	/*pop*/
				self_ 		= ws;	/*pop*/

				/* avoid extra cycle for test cases without test teardowns */
				if (self->tearDown && stateTearDown == self->state )
				{
					break;
				}
				/* do not go through next case while in this state ! */
				else if ( stateTearDown != self->state)
				{
					break;
				}
			}
			else
			{
				/*No testcase ??*/

				self->state = stateTearDown;
			}

		}
		case stateTearDown:
		{
			if (self->tearDown)
			{
				TestResult 	*wr = result_;	/*push*/
				TestCase *ws = self_;	/*push*/

				result_ 	= result;
				self_ 		= self;
				TestListener_doLog(result->listener, self, 0,0,0,utProf_Ev_TestTearDown_Start);
				switch(self->tearDown())
				{
					case ut_BUSY:
						break;
					case ut_DONE:
						self->state = stateEnd;
						break;
					case ut_ABORT:
						self->state = stateEnd;

						TestListener_doLog(result->listener, self, 0,0,0,utProf_Ev_Abort);
						self->abort = 1;
						break;
				}
				TestListener_doLog(result->listener, self, 0,0,0,utProf_Ev_TestTearDown_End);

				result_ 	= wr;	/*pop*/
				self_ 		= ws;	/*pop*/

				if(stateEnd != self->state)
				{
					break;
				}

			}
			else
			{
				self->state = stateEnd;
			}

		}
		case stateEnd:
		{
			TestResult_endTest(result, (Test *)self);
			self->state = stateDefault;
		}
		case stateDefault :
		default :
		{
			self->state = stateDefault;
			/*TestDone - informational*/
		}
	}

}

int TestCase_countTestCases(TestCase *self)
{
	return 1;
}

const TestImplement TestCaseImplement =
{
	(TestNameFunction)			TestCase_name,
	(TestRunFunction)			TestCase_run,
	(TestCountTestCasesFunction)TestCase_countTestCases,
};

void addFailure(const char *msg, unsigned long line, const char *file)
{
	TestResult_addFailure(result_, (Test *)self_, (char *)msg, line, (char *)file);
}

/*
 * Author: 		B&R
 * Added: 		October   09, 2012
*/
void addPassed(const char *msg, unsigned long line, const char *file)
{
	TestResult_addPassed(result_, (Test *)self_, (char *)msg, line, (char *)file);
}

/*
 * Author: 		B&R
 * Added: 		October   23, 2012
*/
void addInfo(const char *msg, unsigned long line, const char *file)
{
	TestResult_addInfo(result_, (Test *)self_, (char *)msg, line, (char *)file);
}

void addAbort(const char *msg, unsigned long line, const char *file)
{
	TestResult_addAbort(result_, (Test *)self_, (char *)msg, line, (char *)file);
}
```

#### profiling.h
```c
#define LOG_DATA(ident, event, addData)  /*	prLog.enable = 1; prLog.objIdent = (unsigned long)ident; prLog.userEvent = event; prLog.pAddData = addData; prLog.addDataLen = stdimpl_strlen(addData); LogEvent(&prLog);*/
```

#### utRunnerTestSuite.c - init cylcic exit handlers
```c
/********************************************************************
 * COPYRIGHT --
 ********************************************************************
 * Program: -
 * Author:
 * Created: August 14, 2012
 ********************************************************************
 * Test registration and handshake
 ********************************************************************/

#include <bur/plctypes.h>

#ifdef _DEFAULT_INCLUDES
#include <AsDefault.h>
#endif

#include "include/utRunner.h"
#include "UtMgr.h"

/* ******************************/
/* TODO: this should be handled by the TestSuite Interface and not with 2 more variables...*/
extern TestSetActive utTestSets[];
extern TestSetList setList;

/* ******************************/

/* Enables this programs test - function pointer called by TestRunnerWebServiceHandler() */
unsigned short run_this_test(UtMgrTestSuite_typ *TestSuiteRef)
{
	switch(TestSuiteRef->Internal.TestHelper.CurrentPhase)
	{
		case utMgrTEST_PHASE_IDLE :
			{	/* Uupdating in idle state (program re-transferred ...) */

				/* Note: Accessing .Interal hurts the API definition a bit, but this code acts as helper for UtMgrTestSuite  in the program's context*/
				TestSuiteRef->Internal.TestHelper.TestSets = (UDINT)setList.list;
				TestSuiteRef->Internal.TestHelper.TestSetCount = setList.nrOfTestSets;
				TestSuiteRef->Internal.TestHelper.CurrentPhase = utMgrTEST_PHASE_RUNNING;
				return ut_BUSY;
			}
		case utMgrTEST_PHASE_RUNNING :
			{
				TestSetActive *locTestSet = (TestSetActive *)TestSuiteRef->Internal.TestHelper.TestSets;
				if(locTestSet[TestSuiteRef->Internal.TestHelper.CurrentTestSet].active)
				{
					switch(UtMgrTestRunnerRunTest((unsigned long)locTestSet[TestSuiteRef->Internal.TestHelper.CurrentTestSet].set))
					{
						case ut_BUSY :
							break;
						case ut_DONE :
						case ut_ABORT:
						default:
							/* goto next test set */
							TestSuiteRef->Internal.TestHelper.CurrentTestSet += 1;
							break;
					}
				}
				else
				{
					TestSuiteRef->Internal.TestHelper.CurrentTestSet++;
				}

				if(TestSuiteRef->Internal.TestHelper.CurrentTestSet >= TestSuiteRef->Internal.TestHelper.TestSetCount)
				{
					TestSuiteRef->Internal.TestHelper.CurrentTestSet = 0;
					TestSuiteRef->Internal.TestHelper.CurrentPhase = utMgrTEST_PHASE_DONE;
				}
				return ut_BUSY;
			}
		case utMgrTEST_PHASE_DONE :
			{
				TestSuiteRef->Internal.TestHelper.CurrentPhase = utMgrTEST_PHASE_IDLE;
				return ut_DONE;
			}
	}
	/* Error occured ...PF?  No specific handling at the moment*/
	return ut_ABORT;
}

	/* Registers Test  */
void utInit(UtMgrTestSuite_typ *TestSuiteRef)
{
	TestSuiteRef->Type = utMgrTEST_TYPE_C;
	TestSuiteRef->Enable = 1;
	/* Note: Accessing .Interal hurts the API definition a bit, but this code acts as helper for UtMgrTestSuite  in the program's context*/
	TestSuiteRef->Internal.TestHelper.TestSets = (UDINT)setList.list;
	TestSuiteRef->Internal.TestHelper.TestSetCount = setList.nrOfTestSets;
	UtMgrTestSuite(TestSuiteRef);
}

void utCyclic(UtMgrTestSuite_typ *TestSuiteRef)
{
	UtMgrTestSuite(TestSuiteRef);
	if(TestSuiteRef->TestActive)
	{
		/* The test code runs in programs own context / task class */
		switch(run_this_test(TestSuiteRef))
		{
			case ut_BUSY :
				break;
			case ut_DONE :
				TestSuiteRef->TestFinished = 1;
				break;
			case ut_ABORT :
			default :
				TestSuiteRef->TestAborted = 1;
		}
	}
	else if (TestSuiteRef->TestFinishedAck)
	{
		TestSuiteRef->TestFinished = 0;
		TestSuiteRef->TestAborted = 0;
	}
}

void  utExit(UtMgrTestSuite_typ *TestSuiteRef)
{
	/* Unregisters Test */
	TestSuiteRef->Enable = 0;
	do
	{
		UtMgrTestSuite(TestSuiteRef);
	}
	while(TestSuiteRef->Busy);
}
```

#### utOther.h
```c
#ifndef	__UT_OTHER_H__
#define	__UT_OTHER_H__

typedef enum utProfEnum
{
    utProf_Ev_Start = 0 /*profUSER_EVENT_START*/ ,
    utProf_Ev_Stop = 1 /*profUSER_EVENT_STOP*/,
    utProf_Ev_MsgFail = 2,
    utProf_Ev_MsgInfo,
    utProf_Ev_MsgPass,
    utProf_Ev_MsgAbort,
    utProf_Ev_Abort,
	utProf_Ev_Skipped,

    utProf_Ev_SetSetup_Start = 20,
    utProf_Ev_SetSetup_End,
    utProf_Ev_SetTearDown_Start,
    utProf_Ev_SetTearDown_End,
    utProf_Ev_SetCylic_Start,
    utProf_Ev_SetCylic_End,
    utProf_Ev_Suite_Start,
    utProf_Ev_Suite_End,
    utProf_Ev_Name_Set_Start,
    utProf_Ev_Name_Set_End,
    /* Testcase, TestSetup , TestTearDown -- "fixture context" */
    utProf_Ev_Fixture_Start,
    utProf_Ev_Fixture_End,
    utProf_Ev_Name_Test_Start,
    utProf_Ev_Name_Test_End,
    utProf_Ev_TestSetup_Start,
    utProf_Ev_TestSetup_End,
    utProf_Ev_TestTearDown_Start,
    utProf_Ev_TestTearDown_End,
    utProf_Ev_TestCase_Start,
    utProf_Ev_TestCase_End,

} utProfEnum;

#endif/*__UT_OTHER_H__*/
```

- Visualisation Logical/mappView (not shown)

Listed in the project but not available here: Logical/Global.typ, Logical/Global.var, Logical/UnitTest/utTrakCtrl/utTrakCtrl/testSuite.c, Logical/UnitTest/Libraries/UnitTest/include
